// TIA Portal V18 export
TYPE "UDT_BoilerUnitState"
// stored: IsFailsafeCompliant false
   STRUCT
      iBoilerSimpleState : Array[1..2] of Int;   // 0-Off, 1 - Heating, 2 - Alarm
      xBoilerOATRequest : Array[1..2] of Bool;
      xBoilerRequestedByAlarm : Array[1..2] of Bool;
      cTarget : Array[1..2] of Byte;
      cActual : Array[1..2] of Byte;
   END_STRUCT;
END_TYPE
